// TIA Portal V18 export
TYPE "ToolCheck_ShW"
// stored: IsFailsafeCompliant false
   STRUCT
      Q_ToolID : Struct
         _1 : String[254];
         _2 : String[254];
         _3 : String[254];
         _4 : String[254];
         _5 : String[254];
         _6 : String[254];
         _7 : String[254];
         _8 : String[254];
         _9 : String[254];
         _10 : String[254];
      END_STRUCT;
      Result : Int;
   END_STRUCT;
END_TYPE
